TYPE T_CodeMRP : STRING[8];
END_TYPE

(* stored: Version 1.1.0.1, ProductVersion 3.1.4024.15
   DUT T_CodeMRP: Id {b8697874-61e4-4e7a-a8c0-f04c4943355c} *)
